Staubli VAL3: setFrameId.pgx

public program setFrameId(num x_nIndex)
begin
  //
end
